INTERFACE ITF_Schuif_DigOutClose_AFO

METHOD set : BOOL
VAR_INPUT
END_VAR
END_METHOD

END_INTERFACE

(* stored: Version 1.1.0.1, ProductVersion 3.1.4026.8
   Itf ITF_Schuif_DigOutClose_AFO: Id {b5089645-feba-46dc-b283-ce020b5b54df}
   Method set: Id {bd492814-0480-47c9-a245-6696c18c92e3} *)
